Staubli VAL3: encodeSharedInt.pgx

public program encodeSharedInt(num& x_nStatus (dimensions=1), num& x_nOutputBuffer[] (dimensions=1), num& x_nBufferPos (dimensions=1), num x_nSharedInt (dimensions=1))
  local num l_nDWordBytes[4]
  local num i
begin
  if x_nStatus<0
    return
  endIf
  x_nStatus=-1
  x_nStatus=toBinary(x_nSharedInt,1,"-4l",l_nDWordBytes)
  if x_nStatus<0
    putln("Failed to encode shared int at index: "+toString("",x_nBufferPos))
    return
  endIf
  call copyArray(x_nOutputBuffer,x_nBufferPos,l_nDWordBytes)
end
